TYPE ST_GantryMachPar :
STRUCT
	Vert_VelocityManual					: LREAL;
	Vert_VelocityAuto					: LREAL;
	Vert_PositionTransport				: LREAL;
	Vert_PositionHome					: LREAL;(* Used when motor is Replaced, write this value as "position bias" in system manager NC-Axis *)
	Vert_PickUpRestPosOffset			: LREAL; // OffsetPosition in which the gantry waits to pickup product from takeout
	
	Hor_VelocityManual					: LREAL;
	Hor_VelocityAuto					: LREAL;
	Hor_PositionHome					: LREAL;(* Used when motor is Replaced, write this value as "position bias" in system manager NC-Axis *)
	PositionHorizontalPickup			: LREAL;
	PositionHorizontalDropOff			: LREAL;

	EnableVacuumSection					: ARRAY [1..6] OF BOOL;
	
	GantryPickupTime					: TIME := T#500MS;
	
	SheetsProduced						: DINT;	// For OEE, total number of sheets produced by this side (A or B).
	ProductsProduced					: DINT; // For OEE, Total number of products produced
	
END_STRUCT
END_TYPE

(* stored: Version 1.1.0.1, ProductVersion 3.1.4020.12
   DUT ST_GantryMachPar: Id {b92b963a-a1a6-4edc-beb7-46e7f395060e} *)
